(* PLC project Unnamed, Unknown Unnamed 1 *)
(* stored: creationDateTime 2023-10-18T21:45:43, modificationDateTime 2023-11-25T00:55:41 *)

PROGRAM program0
  VAR
    Emrg_Stop AT %IX0.0 : BOOL;
    Output_switch AT %IX0.1 : BOOL;
    Gray_water_level AT %IW0.2 : INT := 35;
    Filter_Input_water_level AT %IW0.3 : INT := 35;
    Filter_Output_water_level AT %IW0.4 : INT := 10;
    Clean_water_level AT %IW0.5 : INT := 3;
    Graywater_Pump_RPM AT %IW0.6 : INT;
    Filterwater_Pump_RPM AT %IW0.7 : INT;
    Cleanwater_Pump_RPM AT %IW0.8 : INT;
    Filterwater_Valve AT %QX0.0 : BOOL;
    Cleanwater_Valve AT %QX0.1 : BOOL;
    Filter_inflow_Valve AT %QX0.2 : BOOL;
    Min_Water_Level AT %MW0.0 : INT := 5;
    Max_Water_Level AT %MW0.1 : INT := 25;
    Max_pump_speed AT %MW1.0 : INT := 2000;
    Min_pump_speed AT %MW1.1 : INT := 0;
    Mem1 AT %MW2.0 : BOOL;
    Mem2 AT %MW2.1 : BOOL;
    Mem3 AT %MW2.2 : BOOL;
  END_VAR

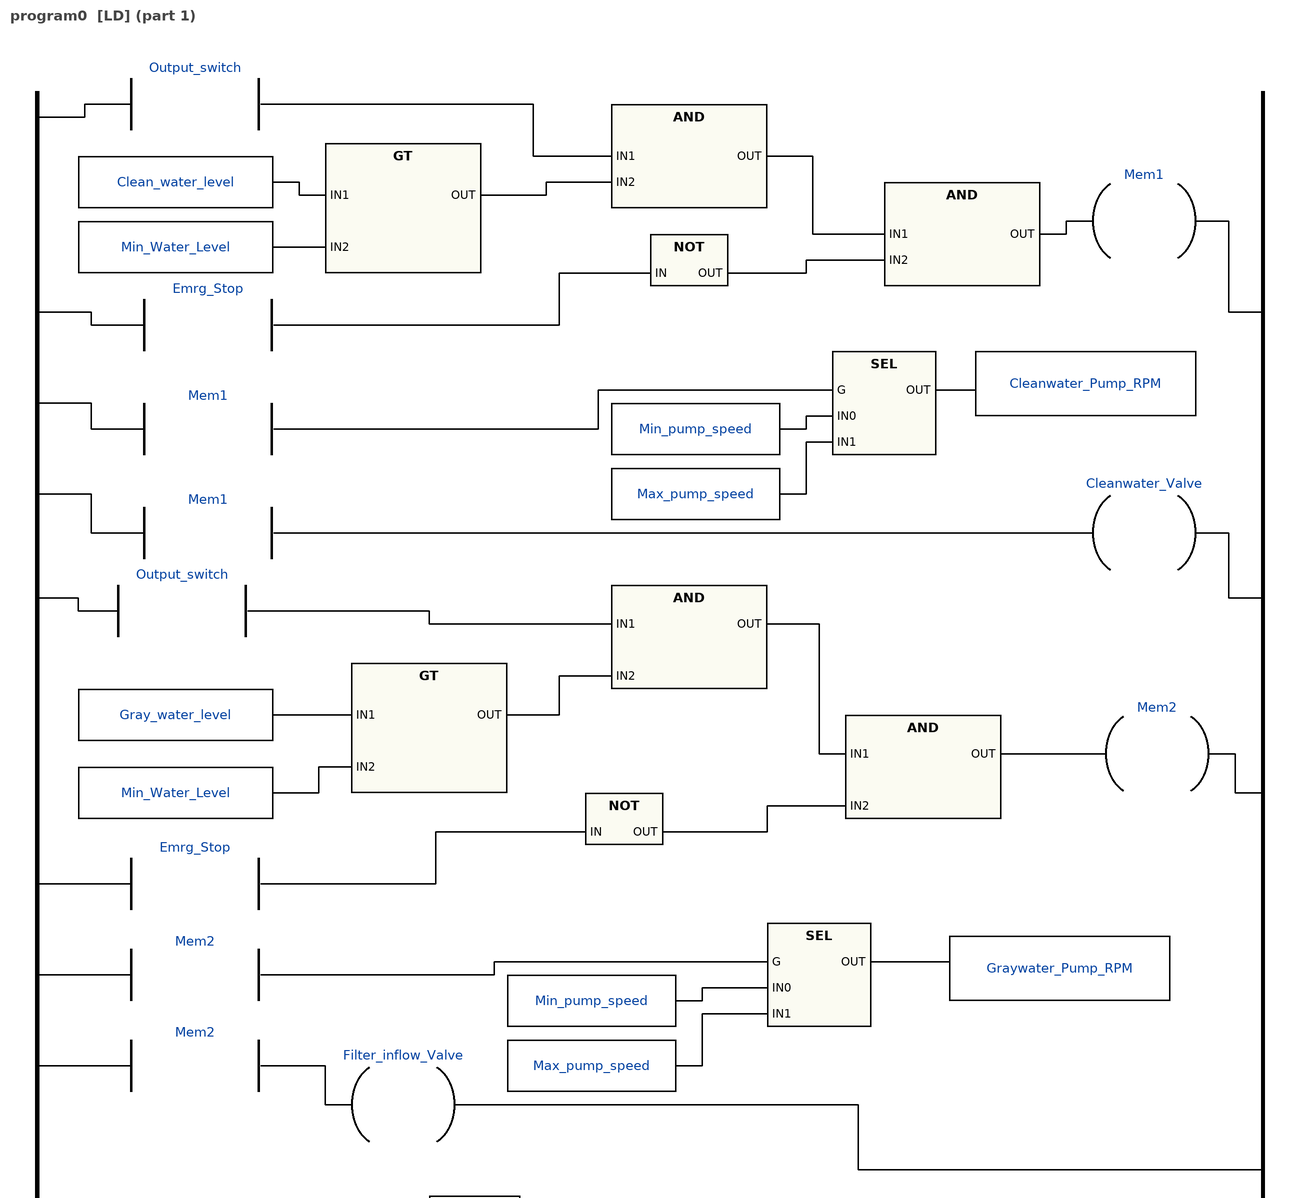
(* LD diagram, written out as Structured Text *)
Mem1 := Output_switch AND Clean_water_level > Min_Water_Level AND NOT Emrg_Stop;
Cleanwater_Pump_RPM := SEL(Mem1, Min_pump_speed, Max_pump_speed);
Cleanwater_Valve := Mem1;
Mem2 := Output_switch AND Gray_water_level > Min_Water_Level AND NOT Emrg_Stop;
Graywater_Pump_RPM := SEL(Mem2, Min_pump_speed, Max_pump_speed);
Filter_inflow_Valve := Mem2;
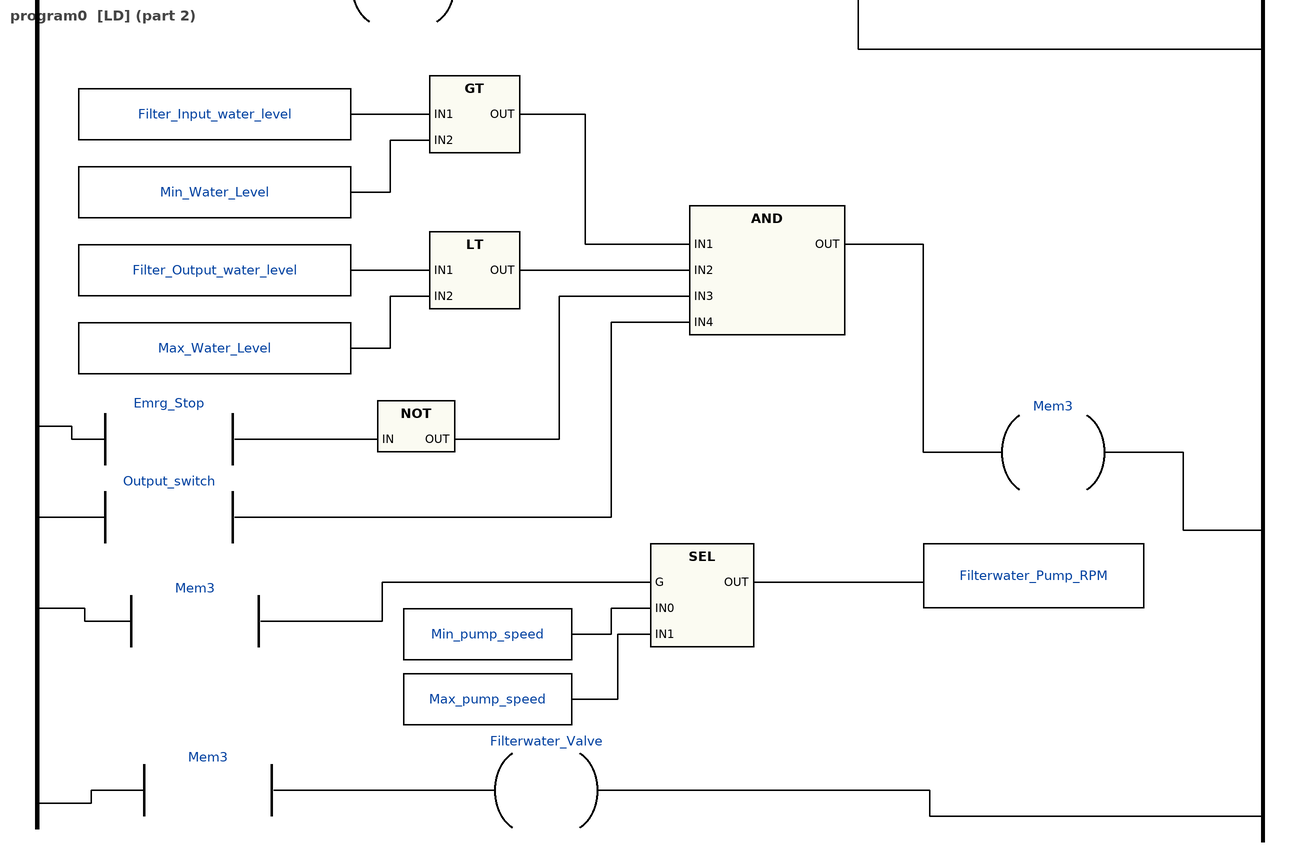
Mem3 := Filter_Input_water_level > Min_Water_Level AND Filter_Output_water_level < Max_Water_Level AND NOT Emrg_Stop AND Output_switch;
Filterwater_Pump_RPM := SEL(Mem3, Min_pump_speed, Max_pump_speed);
Filterwater_Valve := Mem3;
END_PROGRAM

CONFIGURATION Config0
  RESOURCE Res0 ON PLC
    TASK task0(INTERVAL := T#20ms, PRIORITY := 0);
    PROGRAM instance0 WITH task0 : program0;
  END_RESOURCE
END_CONFIGURATION
